// TIA Portal V21 export
VAR_GLOBAL   // PLC tag table "K_TipoTotalizzatore"
END_VAR
VAR_GLOBAL CONSTANT   // user constants
   K_TipoTotalizzatoreDaPortata : Int := 0;
   K_TipoTotalizzatoreDaImpulso : Int := 1;
END_VAR
